FUNCTION_BLOCK FB_ConvStatistic				// Speicher der letzten 10 Rundenzeiten
VAR_INPUT
	vit_LapTime: TIME;						// Input letzter Rundenzeit
END_VAR
VAR_OUTPUT
END_VAR
VAR
	vsi_InPos: INT := 1;					// Zuweisung in welchem Arraybereich die nächste Zeit gespeichert werden soll
	vtt_MaxTime: Time;
END_VAR
VAR_STAT
	vsat_Laps: ARRAY[0..10] OF TIME;		// Deklaration von 10 Speicherplätzen
END_VAR

vsat_Laps[vsi_InPos] := vit_LapTime;		
IF vsi_InPos >= 10 THEN						//falls Array voll, ältester Eintrag überschreiben
	vsi_InPos := 1;							//
ELSE
	vsi_InPos := vsi_InPos +1;				// ansonsten Array 1 hochzählen
END_IF

vtt_MaxTime := FC_GetMaxLapTime(viqat_Laps := vsat_Laps);

END_FUNCTION_BLOCK

(* stored: Version 1.1.0.1
   POU FB_ConvStatistic: Id {43e53574-7e89-46d1-877e-622c34f44f91}, SpecialFunc None *)
